Staubli VAL3: InitVariables.pgx

program InitVariables()
begin
  bAcquisitionStarted = false
  nReceivedByte = 0

  //Dimensions balayage simple
  nScanningLength = 200
  nScanningWidth = 200
  nScanningLineNumber = 20

  //Limites Ref. Cartésien (utiles pour affichage interface graphique)
  nMinHorizontal = -1000
  nMaxHorizontal = 1000
  nMinVertical = -883.44
  nMaxVertical = 950
  nMinRotation = -180
  nMaxRotation = 180


  //Position initiale du robot
  jRobotZeroPosition = {0, 0, 0, 0, 0, 90}
  pRobotZeroPosition = {{50, 50, 950, 0, 0, 0}, {sfree, efree, wfree}}

  //Position initiale de numérisation
  jInitialPosition = {0, 37.32, 99.65, 0, 43.03 ,0}
  pInitialPosition = {{597.67, 50, -72.68, -180, 0, -180}, {sfree, efree, wfree}}

  jInitialPositionRepos = {0, 28.35, 97.17, 0, 54.50, 0}
  pInitialPositionRepos = {{597.67, 50, 27.32,-180,0,-180}, {sfree, efree, wfree}}

  //Position intermédiaire du cercle
  pCircle = pInitialPosition
  pCircle.trsf.x = pCircle.trsf.x - nScanningLength/2
end
